Yaskawa INFORM job: SKRZYNIA_4040_90_STOPNI_10BR.JBI

/JOB
//NAME SKRZYNIA_4040_90_STOPNI_10BR
///FOLDERNAME 02-SKRZYNIE_JOBS
//POS
///NPOS 367,367,0,30,0,0
///TOOL 0
///POSTYPE PULSE
///PULSE
C00000=0,-52280,40443,0,6876,0
C00001=82314,-24956,17040,59626,-27382,6248
C00002=93910,-8625,17040,59626,-43355,6248
C00003=98846,-1061,-42166,80308,-57081,-16120
C00004=100452,6057,-48127,85711,-56704,-21322
C00005=96349,29000,-36127,85072,-63022,-26262
C00006=95580,33075,-33256,84644,-64024,-26851
C00007=94197,33846,-32020,85210,-63413,-26698
C00008=95580,33075,-33256,84644,-64024,-26851
C00009=94888,31114,-36362,85298,-63687,-27185
C00010=95580,33075,-33256,84644,-64024,-26851
C00011=95263,33142,-33256,84677,-63995,-26850
C00012=94634,33491,-32695,84935,-63717,-26781
C00013=94130,33776,-32235,85140,-63494,-26725
C00014=95104,32689,-33981,84829,-63917,-26928
C00015=94679,31503,-35865,85229,-63711,-27129
C00016=95263,33142,-33256,84677,-63995,-26850
C00017=95260,33144,-33256,84678,-63995,-26850
C00018=94650,33483,-32714,84929,-63727,-26783
C00019=94112,33789,-32223,85148,-63489,-26723
C00020=95084,32644,-34054,84845,-63909,-26937
C00021=94657,31449,-35950,85247,-63703,-27139
C00022=95260,33144,-33256,84678,-63995,-26850
C00023=95258,33145,-33257,84676,-63996,-26846
C00024=94953,33314,-32988,84801,-63862,-26812
C00025=94037,33833,-32158,85174,-63457,-26709
C00026=94978,32352,-34521,84941,-63860,-26983
C00027=94597,31295,-36193,85297,-63678,-27162
C00028=95258,33145,-33257,84676,-63996,-26846
C00029=95131,23090,-19879,77391,-65837,-18373
C00030=95120,22557,-18256,76776,-66108,-17621
C00031=94020,23265,-17262,77036,-65497,-17484
C00032=95120,22557,-18256,76776,-66108,-17621
C00033=94446,20406,-21237,77153,-65637,-17798
C00034=95120,22557,-18256,76776,-66108,-17621
C00035=95258,25631,32269,66559,-75499,-2416
C00036=95045,25799,32513,66531,-75379,-2372
C00037=94321,26382,33365,66429,-74973,-2219
C00038=95048,24784,31042,66584,-75290,-2483
C00039=94601,23046,28557,66633,-74859,-2609
C00040=95258,25631,32269,66559,-75499,-2416
C00041=98976,20539,9939,91612,-77544,-12443
C00042=98663,19916,6255,96113,-78269,-14194
C00043=97696,20512,7070,96235,-77611,-14191
C00044=98663,19916,6255,96113,-78269,-14194
C00045=98223,18195,3936,96233,-78026,-14357
C00046=98663,19916,6255,96113,-78269,-14194
C00047=97427,28150,42411,98154,-74759,-5932
C00048=97263,29860,47728,98172,-74140,-4881
C00049=96724,30318,48431,98088,-73756,-4848
C00050=97263,29860,47728,98172,-74140,-4881
C00051=96934,28259,45288,98260,-74017,-5126
C00052=97263,29860,47728,98172,-74140,-4881
C00053=94584,-1413,-17679,107543,-63249,-17346
C00054=98313,-6448,-37250,118963,-73755,-22159
C00055=78553,-42873,-65341,123231,-58560,-22541
C00056=78553,-42984,-66830,123659,-59131,-22943
C00057=97528,-2571,-34675,119478,-73963,-22751
C00058=99837,29570,44224,93766,-77824,-5891
C00059=98826,26629,36097,93853,-77239,-6316
C00060=97856,27338,37141,93774,-76562,-6265
C00061=98826,26629,36097,93853,-77239,-6316
C00062=98480,25016,33743,93919,-77053,-6522
C00063=98826,26629,36097,93853,-77239,-6316
C00064=98236,-3223,-2089,95569,-57848,-9600
C00065=99665,-7201,-6146,95388,-58784,-9416
C00066=48287,-55324,-44178,47560,-5470,10915
C00067=48287,-44591,-17414,16172,-14532,25809
C00068=85348,-13130,13838,41209,-47455,8220
C00069=99199,18818,35660,68259,-73735,-6208
C00070=95720,15423,18785,70454,-68603,-10022
C00071=95720,15423,18785,70454,-68603,-10022
C00072=97055,28839,36684,71776,-79389,-10554
C00073=95990,29701,37981,71658,-78759,-10350
C00074=97107,29731,38027,71793,-79947,-10506
C00075=96750,29830,38178,71892,-80905,-10618
C00076=97107,29731,38027,71793,-79947,-10506
C00077=97055,28839,36684,71776,-79389,-10554
C00078=97055,28839,36684,71776,-79389,-10554
C00079=96028,29668,37934,71662,-78782,-10355
C00080=97055,28839,36684,71776,-79389,-10554
C00081=96569,26658,33449,71833,-78910,-10776
C00082=97055,28839,36684,71776,-79389,-10554
C00083=97055,28839,36684,71776,-79389,-10554
C00084=97055,28839,36684,71776,-79389,-10554
C00085=96073,29634,37879,71669,-78808,-10363
C00086=97055,28839,36684,71776,-79389,-10554
C00087=96556,26588,33346,71835,-78895,-10784
C00088=97055,28839,36684,71776,-79389,-10554
C00089=98688,24309,19320,80205,-78471,-15843
C00090=97055,28839,36684,71776,-79389,-10554
C00091=96070,29634,37881,71667,-78806,-10365
C00092=97055,28839,36684,71776,-79389,-10554
C00093=96542,26531,33264,71837,-78884,-10788
C00094=97055,28839,36684,71776,-79389,-10554
C00095=99365,31341,48046,89916,-78663,6818
C00096=99073,32081,50196,92103,-78109,9106
C00097=98192,32828,51372,91957,-77498,9198
C00098=99073,32081,50196,92103,-78109,9106
C00099=98754,30342,47494,92168,-77945,8838
C00100=99073,32081,50196,92103,-78109,9106
C00101=99780,4859,-8097,97657,-68809,-987
C00102=97427,-15161,-48802,114933,-63377,-9928
C00103=58629,-63760,-77671,121137,-32820,-9668
C00104=58629,-61479,-68873,115361,-30519,-6465
C00105=99951,-8451,-34696,112012,-62700,-7410
C00106=99840,9300,10356,88107,-67494,6780
C00107=99532,23468,17388,90363,-79729,4530
C00108=98411,24191,18413,90419,-78957,4585
C00109=99532,23468,17388,90363,-79729,4530
C00110=99197,22008,15342,90436,-79518,4380
C00111=99532,23468,17388,90363,-79729,4530
C00112=99181,28193,42168,91916,-77030,2884
C00113=98696,27952,42277,91826,-76680,2991
C00114=97999,28483,43076,91734,-76199,3043
C00115=98696,27952,42277,91826,-76680,2991
C00116=98413,26578,40229,91881,-76520,2806
C00117=98696,27952,42277,91826,-76680,2991
C00118=97580,27630,40848,98508,-75244,1367
C00119=97580,27630,40848,98508,-75244,1367
C00120=96916,28152,41628,98436,-74775,1393
C00121=97580,27630,40848,98508,-75244,1367
C00122=97284,26265,38823,98576,-75120,1175
C00123=97580,27630,40848,98508,-75244,1367
C00124=99733,13297,3830,102164,-74334,-5956
C00125=98571,-14980,-17267,89913,-51486,-3548
C00126=44618,-53328,-38563,-7720,-11978,41868
C00127=44299,-51091,-32799,-7549,-14278,41753
///LIMIT ON
C00128=42729,-66511,10542,-1460,2814,7972
C00129=39797,-63802,12228,-1730,2225,8862
///LIMIT OFF
C00130=0,-43112,23163,-32261,-40956,-29092
C00131=50509,-19000,10610,51503,-15997,-61182
C00132=51153,-18191,11234,52953,-16222,-61812
C00133=49506,-16603,12499,51322,-15186,-61219
C00134=50699,-16390,12671,53298,-15774,-62041
C00135=50704,-18403,11069,52157,-16018,-61478
C00136=50704,-18403,11069,52157,-16018,-61478
C00137=51011,-18259,11181,52703,-16157,-61707
C00138=49372,-16676,12437,51065,-15128,-61110
C00139=50855,-16321,12727,53567,-15849,-62152
C00140=50704,-18403,11069,52157,-16018,-61478
C00141=50704,-18403,11069,52157,-16018,-61478
C00142=51194,-17966,11787,52443,-16367,-61556
C00143=49641,-16469,12982,50879,-15396,-60984
C00144=51159,-16110,13274,53409,-16135,-62034
C00145=51194,-19029,8982,55593,-15729,-63095
C00146=51005,-17995,11387,52847,-16122,-61778
C00147=51030,-17982,11395,52891,-16135,-61798
C00148=49666,-16664,12446,51542,-15278,-61306
C00149=51234,-16283,12753,54139,-16047,-62382
C00150=51030,-17982,11395,52891,-16135,-61798
C00151=51030,-17982,11395,52891,-16135,-61798
C00152=51056,-17951,11420,52949,-16145,-61823
C00153=49507,-16445,12622,51407,-15172,-61259
C00154=51212,-15994,12989,54262,-16005,-62444
C00155=51056,-17951,11420,52949,-16145,-61823
C00156=50945,-18019,11363,52741,-16103,-61737
C00157=51451,-18380,9957,55416,-15976,-62984
C00158=49638,-16617,11364,53777,-14815,-62399
C00159=51249,-16205,11700,56405,-15635,-63491
C00160=50945,-18019,11363,52741,-16103,-61737
C00161=50945,-18019,11363,52741,-16103,-61737
C00162=51751,-18888,8325,57986,-15754,-64205
C00163=49901,-17096,9744,56519,-14545,-63700
C00164=51443,-16713,10055,58931,-15359,-64698
C00165=50945,-18019,11363,52741,-16103,-61737
C00166=50945,-18019,11363,52741,-16103,-61737
C00167=51752,-17629,11670,54137,-16475,-62321
C00168=49778,-15710,13222,52239,-15234,-61634
C00169=51536,-15216,13634,55124,-16102,-62830
C00170=50945,-18019,11363,52741,-16103,-61737
C00171=50028,-22953,-3957,22347,-31919,-54220
C00172=50556,-22259,-3444,23037,-31901,-54554
C00173=48685,-20311,-1961,21193,-31011,-53711
C00174=50316,-19877,-1623,23110,-31344,-54618
C00175=49456,-22793,-3840,21729,-31736,-53932
C00176=49763,-25421,-36239,24565,-26935,-60445
C00177=49763,-25421,-36239,24565,-26935,-60445
C00178=47682,-22631,-34091,22709,-25786,-59390
C00179=49411,-21994,-33587,24802,-26153,-60557
C00180=49763,-25421,-36239,24565,-26935,-60445
C00181=50713,-12366,-58367,41124,-17813,-74400
C00182=50531,-11018,-57111,41258,-17631,-74434
C00183=49339,-9106,-55286,40470,-17030,-73839
C00184=50327,-8799,-54988,41498,-17395,-74518
C00185=50078,-11370,-57441,40744,-17481,-74102
C00186=49763,-25421,-36239,24565,-26935,-60445
C00187=49426,-25689,-5908,21254,-32432,-53672
C00188=45389,-28224,4312,35967,-15579,-54278
C00189=40154,-51179,-915,24203,-8234,-36524
C00190=0,-52280,40443,0,6876,0
C00191=21882,-20913,35982,82443,-51729,-53498
C00192=-23487,-14810,34938,67734,-39470,-58782
C00193=1657,-52280,40443,-304,6876,209
C00194=80083,-25473,16734,55938,-25627,7512
C00195=92674,-9533,16184,58080,-41894,6874
C00196=98391,-2369,-43566,80825,-55961,-16033
C00197=100022,4785,-49618,86526,-55706,-21348
C00198=95373,33537,-36121,86560,-63232,-28029
C00199=93881,36038,-32437,85059,-64562,-27761
C00200=93867,33044,-30650,83528,-64743,-25992
C00201=94930,31411,-33227,84334,-64171,-26252
C00202=94930,31411,-33227,84334,-64171,-26252
C00203=93474,31409,-33627,85103,-63552,-26381
C00204=93474,31409,-33627,85103,-63552,-26381
C00205=96539,31728,-33125,83558,-64961,-26367
C00206=95609,19235,-3385,72159,-68881,-11456
C00207=93675,20756,-1492,72153,-69304,-11461
C00208=93706,20835,-1296,72059,-69329,-11411
C00209=95041,22056,296,71883,-70234,-11460
C00210=95041,22056,296,71883,-70234,-11460
C00211=93716,20674,-1606,72153,-69328,-11471
C00212=93749,20787,-1450,72141,-69355,-11463
C00213=95041,22056,296,71883,-70234,-11460
C00214=95041,22056,296,71883,-70234,-11460
C00215=93853,20645,-1646,72134,-69414,-11487
C00216=93701,20690,-1585,72152,-69318,-11471
C00217=95606,21673,-233,71830,-70568,-11545
C00218=95936,-8790,-36169,76308,-52611,-10237
C00219=87381,-35372,-46042,66676,-50803,-1891
C00220=84950,-62287,8062,38288,-37295,1216
C00221=1657,-52280,40443,-304,6876,209
C00222=1657,-52280,40443,-304,6876,209
C00223=-4811,-36310,24637,-49210,-33845,-31988
C00224=41748,-30202,7105,17690,-22932,-42913
C00225=41748,-30202,7105,17690,-22932,-42913
C00226=49037,-21406,10886,33705,-21312,-49933
C00227=57938,-18196,5914,66765,-23183,-68504
C00228=62071,-18819,1330,80566,-26873,-76175
C00229=48249,-23742,8050,33819,-21114,-50004
C00230=-4811,-36310,24637,-49210,-33845,-31988
C00231=1657,-52280,40443,-304,6876,209
C00232=1613,-52280,40443,-296,6876,203
C00233=73560,-62084,7826,28695,-34737,3666
C00234=88377,-34186,-45291,67238,-52212,-2442
C00235=96528,-7533,-34932,76119,-53878,-10439
C00236=100432,21324,12575,83706,-77956,-7498
C00237=98573,22459,14150,83808,-76714,-7352
C00238=97947,26162,19403,83388,-79252,-7038
C00239=97765,26055,19247,83403,-79128,-7046
C00240=99338,18438,8643,84272,-74238,-7648
C00241=98912,19503,1370,96695,-78255,-12346
C00242=97381,18031,1012,96808,-77106,-12025
C00243=97381,18801,8446,95887,-76370,-9901
C00244=100328,20132,10252,95491,-78302,-9647
C00245=98154,32660,54986,101992,-72792,-1753
C00246=94873,38042,64057,104358,-72377,-1226
C00247=94755,38516,64855,104290,-72246,-1148
C00248=94753,45242,81749,102352,-70375,1916
C00249=96613,30369,38748,107128,-77305,-6302
C00250=98457,3518,-7444,102098,-66291,-11392
C00251=98781,-10331,-34310,114047,-66123,-16914
C00252=78936,-45022,-59687,116093,-50330,-16267
C00253=58820,-39124,10926,53325,-41870,3759
C00254=0,-52280,40443,0,6876,0
C00255=0,-36700,24612,-42871,-31823,-33862
C00256=44403,-30110,7154,24155,-23805,-45557
C00257=48366,-23967,9999,33441,-23050,-49710
C00258=57059,-21871,4355,62840,-24072,-66406
C00259=62664,-18498,1251,81512,-27948,-78180
C00260=58407,3196,49521,75767,-22763,-71356
C00261=56068,8902,60102,77374,-19708,-71368
C00262=52721,-13182,18231,110850,-19193,-88536
C00263=47073,-34549,9488,27883,-30316,-51458
C00264=0,-52247,40504,0,6859,0
C00265=41126,-41934,51032,-5894,-46731,13127
C00266=87376,-42070,-11985,58546,-50710,87
C00267=101177,-2604,23124,67435,-62482,198
C00268=97923,11434,18635,75872,-68057,-4429
C00269=99135,26942,27967,80896,-80067,-11
C00270=97959,27246,28410,80885,-79279,71
C00271=97910,25581,20036,81620,-78756,-2039
C00272=99054,25606,22085,82627,-78975,-1891
C00273=98877,27968,32487,76173,-79945,2468
C00274=95369,26181,23160,71095,-76769,901
C00275=95369,28262,32501,70203,-78207,3099
C00276=100802,24456,20984,80151,-80320,-697
C00277=99662,22785,17568,82066,-77607,-1267
C00278=97757,25456,21360,81884,-78797,-1037
C00279=97789,25433,21327,81884,-78819,-1041
C00280=99676,21999,16470,82145,-76972,-1318
C00281=97441,-6012,-18634,86114,-58345,-2339
C00282=92377,-33385,-41303,83059,-36844,1354
C00283=79425,-37128,-15462,51820,-35721,18807
C00284=43180,-50572,-20637,6552,-29302,38834
///LIMIT ON
C00285=37721,-67612,11381,1325,-438,7850
///LIMIT OFF
C00286=37164,-60659,6466,13301,-5027,-19773
C00287=45362,-39990,2831,27538,-17767,-40935
C00288=55315,-20486,12421,43917,-25084,-54085
C00289=61687,-17127,4357,78253,-26449,-75506
C00290=66887,-15221,5723,82563,-32969,-76938
C00291=53534,-30170,6270,37667,-26637,-51098
C00292=41180,-61187,4729,17280,-8498,-23442
C00293=0,-52280,40443,0,6876,0
C00294=0,-52280,40443,0,6876,0
///LIMIT ON
C00295=37721,-67612,11381,1325,-438,7850
///LIMIT OFF
C00296=43180,-50572,-20637,6552,-29302,38834
C00297=79425,-37128,-15462,51820,-35721,18807
C00298=92377,-33385,-41303,83059,-36844,1354
C00299=100252,-4949,-17551,85890,-60241,-2391
C00300=99662,22785,17568,82066,-77607,-1267
C00301=98003,26711,23176,81782,-79695,-932
C00302=98187,26766,23256,81772,-79821,-932
C00303=99662,22785,17568,82066,-77607,-1267
C00304=99662,22785,17568,82066,-77607,-1267
C00305=97671,26258,22515,81825,-79282,-965
C00306=97727,26283,22551,81822,-79321,-966
C00307=99662,22785,17568,82066,-77607,-1267
C00308=99171,25371,27709,97207,-78195,-1592
C00309=97098,23330,25144,97300,-76842,-1817
C00310=97098,25842,34993,96283,-76010,469
C00311=99772,20639,8352,98678,-80464,-6065
C00312=98552,-10425,-57317,115530,-68576,-16387
C00313=72212,-55568,-87372,121854,-47773,-15081
C00314=43180,-50572,-20637,6552,-29302,38834
///LIMIT ON
C00315=37721,-67612,11381,1325,-438,7850
///LIMIT OFF
C00316=0,-52280,40443,0,6876,0
C00317=0,-52280,40443,0,6876,0
///LIMIT ON
C00318=23708,-46776,23536,16027,-4787,-19738
///LIMIT OFF
C00319=50917,-40459,4132,34421,-18173,-42391
C00320=55315,-20486,12421,43917,-25084,-54085
C00321=52021,-27344,-11614,25442,-32756,-51822
C00322=62388,-19076,-7315,47741,-37100,-57915
C00323=60492,-23043,-43968,60514,-28343,-68592
C00324=52021,-27344,-11614,25442,-32756,-51822
C00325=50917,-40459,4132,34421,-18173,-42391
C00326=56351,-28617,-8977,50177,-24220,-59041
C00327=61013,-25727,-20437,91852,-25479,-87385
C00328=68741,-23000,-19911,95900,-36007,-87783
C00329=59870,-32730,-20784,77712,-26701,-76039
C00330=36994,-41399,-15582,14937,-21377,-43241
C00331=31287,-69981,-10850,7253,-6843,-20996
C00332=19644,-57271,30737,863,5243,-2499
C00333=0,-52280,40443,0,6876,0
C00334=0,-52280,40443,0,6876,0
///LIMIT ON
C00335=37721,-67612,11381,1325,-438,7850
///LIMIT OFF
C00336=43180,-50572,-20637,6552,-29302,38834
C00337=92325,-17806,9716,57334,-44195,17168
C00338=83562,-2075,23934,52242,-47081,17120
C00339=81926,-4528,18929,54087,-44625,16400
C00340=98156,27605,40467,74304,-79249,6093
C00341=97389,28448,36068,78537,-79231,3814
C00342=97907,24801,21502,85617,-78711,-660
C00343=99547,21785,17244,85874,-76675,-945
C00344=99107,21615,15088,95660,-77501,-3171
C00345=97330,21661,23948,94493,-75452,-401
C00346=97330,25174,37197,92971,-74702,2673
C00347=100285,22853,27662,91564,-77234,921
C00348=95045,29770,44207,110893,-72615,-445
C00349=92602,30098,46290,110515,-70628,-245
C00350=91321,34137,56434,112423,-68257,619
C00351=92127,32273,50247,113174,-70001,-486
C00352=99547,27249,39584,83596,-77197,4391
C00353=85644,-16652,-26140,89995,-40279,-1638
C00354=96357,-21723,-30363,88205,-47532,-883
C00355=98913,1421,32623,59426,-59934,14740
C00356=68865,-35989,-5252,49829,-38105,21179
C00357=80632,-38079,-20908,64053,-45216,12949
C00358=43180,-50572,-20637,6552,-29302,38834
C00359=50917,-40459,4132,34421,-18173,-42391
C00360=55315,-20486,12421,43917,-25084,-54085
C00361=52609,-18323,14042,41333,-23544,-53138
C00362=70054,-15959,-1295,94448,-37577,-86566
C00363=61757,-17157,6384,73937,-27308,-72117
C00364=37618,-28118,7425,14704,-21495,-41826
C00365=31287,-69981,-10850,7253,-6843,-20996
C00366=0,-52280,40443,0,6876,0
BC00000=376110
BC00001=352964
BC00002=352964
BC00003=352964
BC00004=352964
BC00005=352964
BC00006=352964
BC00007=352964
BC00008=352964
BC00009=352964
BC00010=352964
BC00011=399066
BC00012=399066
BC00013=399066
BC00014=399066
BC00015=399066
BC00016=399066
BC00017=445276
BC00018=445276
BC00019=445276
BC00020=445276
BC00021=445276
BC00022=445276
BC00023=491380
BC00024=491380
BC00025=491380
BC00026=491380
BC00027=491380
BC00028=491380
BC00029=477558
BC00030=476336
BC00031=476336
BC00032=476336
BC00033=476336
BC00034=476336
BC00035=467227
BC00036=467227
BC00037=467227
BC00038=467227
BC00039=467227
BC00040=467227
BC00041=479694
BC00042=482001
BC00043=482001
BC00044=482001
BC00045=482001
BC00046=482001
BC00047=469388
BC00048=468082
BC00049=468082
BC00050=468082
BC00051=468082
BC00052=468082
BC00053=467166
BC00054=467166
BC00055=467166
BC00056=581600
BC00057=581600
BC00058=528199
BC00059=528202
BC00060=528202
BC00061=528202
BC00062=528202
BC00063=528202
BC00064=531560
BC00065=531560
BC00066=512089
BC00067=606955
BC00068=621951
BC00069=621951
BC00070=621951
BC00071=621951
BC00072=621951
BC00073=621951
BC00074=621951
BC00075=621951
BC00076=621951
BC00077=645037
BC00078=645037
BC00079=645037
BC00080=645037
BC00081=645037
BC00082=645037
BC00083=691109
BC00084=691109
BC00085=691109
BC00086=691109
BC00087=691109
BC00088=691109
BC00089=714197
BC00090=714197
BC00091=714197
BC00092=714197
BC00093=714197
BC00094=714197
BC00095=704400
BC00096=703157
BC00097=703157
BC00098=703157
BC00099=703157
BC00100=703157
BC00101=703157
BC00102=713115
BC00103=713115
BC00104=805551
BC00105=805551
BC00106=781418
BC00107=793824
BC00108=793824
BC00109=793824
BC00110=793824
BC00111=793824
BC00112=808984
BC00113=808984
BC00114=808984
BC00115=808984
BC00116=808984
BC00117=808984
BC00118=829368
BC00119=829368
BC00120=829368
BC00121=829368
BC00122=829368
BC00123=829368
BC00124=829627
BC00125=821657
BC00126=814103
BC00127=795686
BC00128=693498
BC00129=688280
BC00130=719629
BC00131=797458
BC00132=797458
BC00133=797458
BC00134=797458
BC00135=797458
BC00136=736016
BC00137=736016
BC00138=736016
BC00139=736016
BC00140=736016
BC00141=674586
BC00142=674586
BC00143=674586
BC00144=674586
BC00145=674586
BC00146=613184
BC00147=613184
BC00148=613184
BC00149=613184
BC00150=613184
BC00151=555022
BC00152=555022
BC00153=555022
BC00154=555022
BC00155=555022
BC00156=490298
BC00157=490298
BC00158=490298
BC00159=490298
BC00160=490298
BC00161=428826
BC00162=428826
BC00163=428826
BC00164=428826
BC00165=428826
BC00166=367374
BC00167=367374
BC00168=367374
BC00169=367374
BC00170=367374
BC00171=367378
BC00172=367378
BC00173=367378
BC00174=367378
BC00175=367378
BC00176=367378
BC00177=367378
BC00178=367378
BC00179=367378
BC00180=367378
BC00181=367378
BC00182=367378
BC00183=367378
BC00184=367378
BC00185=367378
BC00186=367378
BC00187=367378
BC00188=367374
BC00189=441050
BC00190=441050
BC00191=743708
BC00192=782128
BC00193=352964
BC00194=352964
BC00195=352964
BC00196=406723
BC00197=352964
BC00198=352964
BC00199=352964
BC00200=353556
BC00201=353556
BC00202=391964
BC00203=400107
BC00204=389591
BC00205=400107
BC00206=381081
BC00207=388817
BC00208=381081
BC00209=388818
BC00210=427169
BC00211=434877
BC00212=427169
BC00213=427169
BC00214=450237
BC00215=457913
BC00216=450237
BC00217=450041
BC00218=450041
BC00219=450041
BC00220=450041
BC00221=450041
BC00222=400994
BC00223=490644
BC00224=563016
BC00225=563016
BC00226=563016
BC00227=563016
BC00228=624476
BC00229=624476
BC00230=490644
BC00231=400994
BC00232=402304
BC00233=450041
BC00234=450041
BC00235=498778
BC00236=451598
BC00237=451598
BC00238=459362
BC00239=451598
BC00240=459288
BC00241=484574
BC00242=484574
BC00243=484574
BC00244=484574
BC00245=464718
BC00246=464718
BC00247=464718
BC00248=469790
BC00249=469790
BC00250=467718
BC00251=475246
BC00252=427384
BC00253=476890
BC00254=492251
BC00255=720637
BC00256=795617
BC00257=801528
BC00258=805368
BC00259=808796
BC00260=777283
BC00261=777283
BC00262=777285
BC00263=760893
BC00264=538671
BC00265=564292
BC00266=544905
BC00267=523419
BC00268=548184
BC00269=573245
BC00270=573245
BC00271=573245
BC00272=569148
BC00273=617841
BC00274=629475
BC00275=629475
BC00276=631879
BC00277=634993
BC00278=633229
BC00279=640937
BC00280=640937
BC00281=640937
BC00282=640937
BC00283=640937
BC00284=640937
BC00285=640937
BC00286=469376
BC00287=406602
BC00288=315730
BC00289=315725
BC00290=377231
BC00291=377231
BC00292=431999
BC00293=431999
BC00294=640937
BC00295=640937
BC00296=640937
BC00297=640937
BC00298=640937
BC00299=640937
BC00300=679258
BC00301=679258
BC00302=687013
BC00303=679258
BC00304=702338
BC00305=702338
BC00306=710018
BC00307=702338
BC00308=711372
BC00309=711372
BC00310=711372
BC00311=711372
BC00312=723912
BC00313=723912
BC00314=703131
BC00315=640937
BC00316=640937
BC00317=492251
BC00318=483911
BC00319=372992
BC00320=315730
BC00321=315730
BC00322=315730
BC00323=315730
BC00324=315730
BC00325=421515
BC00326=465804
BC00327=465238
BC00328=526388
BC00329=526326
BC00330=526236
BC00331=526236
BC00332=526236
BC00333=526236
BC00334=640937
BC00335=640937
BC00336=792907
BC00337=785422
BC00338=785422
BC00339=785422
BC00340=808786
BC00341=808610
BC00342=816482
BC00343=816482
BC00344=831767
BC00345=831767
BC00346=831767
BC00347=831767
BC00348=812640
BC00349=812640
BC00350=812640
BC00351=812640
BC00352=814454
BC00353=818927
BC00354=798802
BC00355=772424
BC00356=743273
BC00357=702349
BC00358=657048
BC00359=664515
BC00360=684473
BC00361=684473
BC00362=684473
BC00363=745829
BC00364=745829
BC00365=650116
BC00366=650116
///POSTYPE BASE
///RECTAN
///RCONF 0,0,0,0,0,0,0,0,0,0,0,0,0,0,0,0,0,0,0,0,0,0,0,0
P00006=-2.449,0.031,8.825,0.0000,0.0000,0.0000
P00058=0.000,0.000,3.000,0.0000,0.0000,0.0000
///RCONF 1,0,0,0,0,0,0,0,0,0,0,0,0,0,0,0,0,0,0,0,0,0,0,0
P00300=-0.036,-1.505,2.318,0.0000,0.0000,0.0000
///RCONF 0,0,0,0,0,0,0,0,0,0,0,0,0,0,0,0,0,0,0,0,0,0,0,0
P00301=0.005,-4.708,-4.628,0.0000,0.0000,0.0000
P00302=0.052,-2.937,-4.426,0.0000,0.0000,0.0000
P00303=-0.004,-1.437,-4.584,0.0000,0.0000,0.0000
P00304=0.028,-1.666,-4.234,0.0000,0.0000,0.0000
P00305=-0.003,-1.920,-3.501,0.0000,0.0000,0.0000
P00306=0.015,-2.252,-3.054,0.0000,0.0000,0.0000
P00307=0.019,-2.151,-5.077,0.0000,0.0000,0.0000
P00308=-0.003,-2.092,-4.888,0.0000,0.0000,0.0000
P00309=-0.040,-2.205,-4.992,0.0000,0.0000,0.0000
P00310=-0.006,-2.490,-5.925,0.0000,0.0000,0.0000
P00311=-0.007,-2.079,-5.307,0.0000,0.0000,0.0000
P00312=-0.032,2.202,-7.632,0.0000,0.0000,0.0000
///RCONF 1,0,0,0,0,0,0,0,0,0,0,0,0,0,0,0,0,0,0,0,0,0,0,0
P00313=-0.088,1.055,2.110,0.0000,0.0000,0.0000
P00314=-0.055,1.752,1.634,0.0000,0.0000,0.0000
P00316=0.009,2.112,2.075,0.0000,0.0000,0.0000
P00317=-0.015,2.781,3.126,0.0000,0.0000,0.0000
///RCONF 0,0,0,0,0,0,0,0,0,0,0,0,0,0,0,0,0,0,0,0,0,0,0,0
P00351=13.563,-0.027,-0.653,0.0000,0.0000,0.0000
P00352=13.252,-0.027,-0.827,0.0000,0.0000,0.0000
P00353=10.971,-0.082,0.776,0.0000,0.0000,0.0000
P00354=-0.024,2.508,-1.824,0.0000,0.0000,0.0000
P00355=-0.001,2.528,-1.131,0.0000,0.0000,0.0000
P00356=-0.034,2.921,-0.262,0.0000,0.0000,0.0000
P00357=0.003,3.386,-0.091,0.0000,0.0000,0.0000
P00358=0.014,3.037,-0.020,0.0000,0.0000,0.0000
P00359=-0.005,2.731,0.912,0.0000,0.0000,0.0000
P00360=-0.011,3.412,0.438,0.0000,0.0000,0.0000
P00361=0.018,3.050,1.253,0.0000,0.0000,0.0000
//INST
///DATE 2025/03/25 09:39
///ATTR SC,RW
///GROUP1 RB1,BS1
NOP
CALL JOB:MOVE_INTO_TUNNEL
MOVJ C00000 BC00000 VJ=50.00
MOVJ C00001 BC00001 VJ=30.00
MOVJ C00002 BC00002 VJ=30.00
COMM MOVL C00003 BC00003 V=333.3
COMM MOVJ C00004 BC00004 VJ=30.00
COMM MOVL C00005 BC00005 V=500.0
COMM '------------------------
COMM 'W31.2
COMM '------------------------
COMM MOVL C00006 BC00006 V=166.7 PL=0
COMM REFP 3 C00007 BC00007
COMM CALL JOB:SEARCH-R1
COMM SET P0300 P0006
COMM SFTON P0300
COMM MOVL C00008 BC00008 V=66.7 PL=0
COMM REFP 3 C00009 BC00009
COMM CALL JOB:SEARCH-R1
COMM SET P0300 P0006
COMM SFTON P0300
COMM MOVL C00010 BC00010 V=166.7 PL=0
COMM SFTOF
COMM '------------------------
COMM 'W31.4
COMM '------------------------
COMM MOVL C00011 BC00011 V=666.7
COMM MOVL C00012 BC00012 V=83.3 PL=0
COMM REFP 3 C00013 BC00013
COMM CALL JOB:SEARCH-R1
COMM SET P0301 P0006
COMM SFTON P0301
COMM MOVL C00014 BC00014 V=166.7 PL=0
COMM REFP 3 C00015 BC00015
COMM CALL JOB:SEARCH-R1
COMM SET P0301 P0006
COMM SFTON P0301
COMM MOVL C00016 BC00016 V=166.7 PL=0
COMM SFTOF
'------------------------
'W31.6
'------------------------
MOVL C00017 BC00017 V=666.7
MOVL C00018 BC00018 V=83.3 PL=0
REFP 3 C00019 BC00019
CALL JOB:SEARCH-R1
SET P0302 P0006
SFTON P0302
MOVL C00020 BC00020 V=166.7 PL=0
REFP 3 C00021 BC00021
CALL JOB:SEARCH-R1
SET P0302 P0006
SFTON P0302
MOVL C00022 BC00022 V=250.0 PL=0
SFTOF
'------------------------
'W31.8
'------------------------
MOVL C00023 BC00023 V=666.7
MOVL C00024 BC00024 V=83.3 PL=0
REFP 3 C00025 BC00025
CALL JOB:SEARCH-R1
SET P0303 P0006
SFTON P0303
MOVL C00026 BC00026 V=166.7 PL=0
REFP 3 C00027 BC00027
CALL JOB:SEARCH-R1
SET P0303 P0006
SFTON P0303
MOVL C00028 BC00028 V=250.0 PL=0
SFTOF
'------------------------
'W31.9
'------------------------
MOVL C00029 BC00029 V=666.7
MOVL C00030 BC00030 V=83.3 PL=0
REFP 3 C00031 BC00031
CALL JOB:SEARCH-R1
SET P0304 P0006
SFTON P0304
MOVL C00032 BC00032 V=166.7 PL=0
REFP 3 C00033 BC00033
CALL JOB:SEARCH-R1
SET P0304 P0006
SFTON P0304
MOVL C00034 BC00034 V=250.0 PL=0
SFTOF
'------------------------
'W31.11
'------------------------
MOVL C00035 BC00035 V=666.7
MOVL C00036 BC00036 V=83.3 PL=0
REFP 3 C00037 BC00037
CALL JOB:SEARCH-R1
SET P0305 P0006
SFTON P0305
MOVL C00038 BC00038 V=166.7 PL=0
REFP 3 C00039 BC00039
CALL JOB:SEARCH-R1
SET P0305 P0006
SFTON P0305
MOVL C00040 BC00040 V=250.0 PL=0
SFTOF
'------------------------
'W31.13
'------------------------
MOVL C00041 BC00041 V=666.7
MOVL C00042 BC00042 V=166.7 PL=0
REFP 3 C00043 BC00043
CALL JOB:SEARCH-R1
SET P0306 P0006
SFTON P0306
MOVL C00044 BC00044 V=166.7 PL=0
REFP 3 C00045 BC00045
CALL JOB:SEARCH-R1
SET P0306 P0006
SFTON P0306
MOVL C00046 BC00046 V=250.0 PL=0
SFTOF
'------------------------
'W31.14
'------------------------
MOVL C00047 BC00047 V=666.7
MOVL C00048 BC00048 V=100.0 PL=0
REFP 3 C00049 BC00049
CALL JOB:SEARCH-R1
SET P0307 P0006
SFTON P0307
MOVL C00050 BC00050 V=166.7 PL=0
REFP 3 C00051 BC00051
CALL JOB:SEARCH-R1
SET P0307 P0006
SFTON P0307
MOVL C00052 BC00052 V=250.0 PL=0
SFTOF
'------------------------
MOVL C00053 BC00053 V=333.3
MOVL C00054 BC00054 V=333.3
MOVL C00055 BC00055 V=333.3
MOVL C00056 BC00056 V=666.7
MOVL C00057 BC00057 V=666.7
'W31.16
'------------------------
MOVL C00058 BC00058 V=666.7
MOVL C00059 BC00059 V=100.0 PL=0
REFP 3 C00060 BC00060
CALL JOB:SEARCH-R1
SET P0308 P0006
SFTON P0308
MOVL C00061 BC00061 V=166.7 PL=0
REFP 3 C00062 BC00062
CALL JOB:SEARCH-R1
SET P0308 P0006
SFTON P0308
MOVL C00063 BC00063 V=250.0 PL=0
SFTOF
MOVL C00064 BC00064 V=666.7
MOVL C00065 BC00065 V=666.7
MOVL C00066 BC00066 V=500.0 PL=1
MOVJ C00067 BC00067 VJ=60.00
MOVL C00068 BC00068 V=833.3 PL=0
MOVL C00069 BC00069 V=500.0 PL=0
MOVL C00070 BC00070 V=500.0 PL=0
'------------------------
'W31.18
'------------------------
MOVL C00071 BC00071 V=333.3 PL=0
SFTOF
MOVL C00072 BC00072 V=133.3 PL=0
REFP 3 C00073 BC00073
CALL JOB:SEARCH-R1
SET P0309 P0006
SFTON P0309
MOVL C00074 BC00074 V=166.7 PL=0
REFP 3 C00075 BC00075
CALL JOB:SEARCH-R1
SET P0309 P0006
SFTON P0309
MOVL C00076 BC00076 V=250.0 PL=0
SFTOF
'------------------------
'W31.19
'------------------------
MOVL C00077 BC00077 V=666.7
MOVL C00078 BC00078 V=100.0 PL=0
REFP 3 C00079 BC00079
CALL JOB:SEARCH-R1
SET P0310 P0006
SFTON P0310
MOVL C00080 BC00080 V=166.7 PL=0
REFP 3 C00081 BC00081
CALL JOB:SEARCH-R1
SET P0310 P0006
SFTON P0310
MOVL C00082 BC00082 V=250.0 PL=0
SFTOF
'------------------------
'W31.21
'------------------------
MOVL C00083 BC00083 V=666.7
MOVL C00084 BC00084 V=100.0 PL=0
REFP 3 C00085 BC00085
CALL JOB:SEARCH-R1
SET P0311 P0006
SFTON P0311
MOVL C00086 BC00086 V=166.7 PL=0
REFP 3 C00087 BC00087
CALL JOB:SEARCH-R1
SET P0311 P0006
SFTON P0311
MOVL C00088 BC00088 V=250.0 PL=0
SFTOF
'------------------------
'W31.22
'------------------------
MOVL C00089 BC00089 V=666.7
MOVL C00090 BC00090 V=100.0 PL=0
REFP 3 C00091 BC00091
CALL JOB:SEARCH-R1
SET P0312 P0006
SFTON P0312
MOVL C00092 BC00092 V=166.7 PL=0
REFP 3 C00093 BC00093
CALL JOB:SEARCH-R1
SET P0312 P0006
SFTON P0312
MOVL C00094 BC00094 V=250.0 PL=0
SFTOF
'------------------------
'W31.24
'------------------------
MOVL C00095 BC00095 V=666.7
MOVL C00096 BC00096 V=100.0 PL=0
REFP 3 C00097 BC00097
CALL JOB:SEARCH-R1
SET P0313 P0006
SFTON P0313
MOVL C00098 BC00098 V=166.7 PL=0
REFP 3 C00099 BC00099
CALL JOB:SEARCH-R1
SET P0313 P0006
SFTON P0313
MOVL C00100 BC00100 V=166.7 PL=0
SFTOF
MOVL C00101 BC00101 V=666.7
MOVL C00102 BC00102 V=666.7
MOVL C00103 BC00103 V=666.7
MOVL C00104 BC00104 V=666.7
MOVL C00105 BC00105 V=666.7
'------------------------
'W31.26
'------------------------
MOVL C00106 BC00106 V=666.7
MOVL C00107 BC00107 V=100.0 PL=0
REFP 3 C00108 BC00108
CALL JOB:SEARCH-R1
SET P0314 P0006
SFTON P0314
MOVL C00109 BC00109 V=166.7 PL=0
REFP 3 C00110 BC00110
CALL JOB:SEARCH-R1
SET P0314 P0006
SFTON P0314
MOVL C00111 BC00111 V=250.0 PL=0
SFTOF
'------------------------
'W31.29
'------------------------
MOVL C00112 BC00112 V=166.7
MOVL C00113 BC00113 V=100.0 PL=0
REFP 3 C00114 BC00114
CALL JOB:SEARCH-R1
SET P0316 P0006
SFTON P0316
MOVL C00115 BC00115 V=166.7 PL=0
REFP 3 C00116 BC00116
CALL JOB:SEARCH-R1
SET P0316 P0006
SFTON P0316
MOVL C00117 BC00117 V=250.0 PL=0
SFTOF
'------------------------
'W31.31
'------------------------
MOVL C00118 BC00118 V=250.0
MOVL C00119 BC00119 V=100.0 PL=0
REFP 3 C00120 BC00120
CALL JOB:SEARCH-R1
SET P0317 P0006
SFTON P0317
MOVL C00121 BC00121 V=166.7 PL=0
REFP 3 C00122 BC00122
CALL JOB:SEARCH-R1
SET P0317 P0006
SFTON P0317
MOVL C00123 BC00123 V=250.0 PL=0
SFTOF
'------------------------
'W31.32
'------------------------
MOVL C00124 BC00124 V=500.0
MOVL C00125 BC00125 V=500.0
MOVL C00126 BC00126 V=500.0
MOVL C00127 BC00127 V=666.7
MOVJ C00128 BC00128 VJ=80.00
MOVJ C00129 BC00129 VJ=80.00
MOVJ C00130 BC00130 VJ=50.00
'------------------------
'W214A L
'------------------------
MOVJ C00131 BC00131 VJ=30.00
MOVL C00132 BC00132 V=100.0 PL=0
REFP 3 C00133 BC00133
CALL JOB:SEARCH-R1
IMOV P0058 V=11.7
SET P0351 P0006
SFTON P0351
REFP 3 C00134 BC00134
CALL JOB:SEARCH-R1
SET P0351 P0006
SFTON P0351
MOVL C00135 BC00135 V=250.0 PL=0
SFTOF
'------------------------
'W219A P
'------------------------
MOVJ C00136 BC00136 VJ=40.00
MOVL C00137 BC00137 V=100.0 PL=0
REFP 3 C00138 BC00138
CALL JOB:SEARCH-R1
IMOV P0058 V=11.7
SET P0352 P0006
SFTON P0352
REFP 3 C00139 BC00139
CALL JOB:SEARCH-R1
SET P0352 P0006
SFTON P0352
MOVL C00140 BC00140 V=250.0 PL=0
SFTOF
'------------------------
'W219A L
'------------------------
MOVJ C00141 BC00141 VJ=50.00
MOVL C00142 BC00142 V=166.7 PL=0
REFP 3 C00143 BC00143
CALL JOB:SEARCH-R1
IMOV P0058 V=11.7
SET P0353 P0006
SFTON P0353
REFP 3 C00144 BC00144
CALL JOB:SEARCH-R1
SET P0353 P0006
SFTON P0353
MOVL C00145 BC00145 V=250.0 PL=0
SFTOF
'------------------------
'W213A P
'------------------------
MOVJ C00146 BC00146 VJ=60.00
MOVL C00147 BC00147 V=166.7 PL=0
REFP 3 C00148 BC00148
CALL JOB:SEARCH-R1
IMOV P0058 V=11.7
SET P0354 P0006
SFTON P0354
REFP 3 C00149 BC00149
CALL JOB:SEARCH-R1
SET P0354 P0006
SFTON P0354
MOVL C00150 BC00150 V=250.0 PL=0
SFTOF
'------------------------
'W213A L
'------------------------
MOVJ C00151 BC00151 VJ=50.00
MOVL C00152 BC00152 V=166.7 PL=0
REFP 3 C00153 BC00153
CALL JOB:SEARCH-R1
IMOV P0058 V=11.7
SET P0355 P0006
SFTON P0355
REFP 3 C00154 BC00154
CALL JOB:SEARCH-R1
SET P0355 P0006
SFTON P0355
MOVL C00155 BC00155 V=250.0 PL=0
SFTOF
'------------------------
'W218A P
'------------------------
MOVJ C00156 BC00156 VJ=60.00
MOVL C00157 BC00157 V=166.7 PL=0
REFP 3 C00158 BC00158
CALL JOB:SEARCH-R1
IMOV P0058 V=11.7
SET P0356 P0006
SFTON P0356
REFP 3 C00159 BC00159
CALL JOB:SEARCH-R1
SET P0356 P0006
SFTON P0356
MOVL C00160 BC00160 V=250.0 PL=0
SFTOF
'------------------------
'W218A L
'------------------------
MOVJ C00161 BC00161 VJ=60.00
MOVL C00162 BC00162 V=166.7 PL=0
REFP 3 C00163 BC00163
CALL JOB:SEARCH-R1
IMOV P0058 V=11.7
SET P0357 P0006
SFTON P0357
REFP 3 C00164 BC00164
CALL JOB:SEARCH-R1
SET P0357 P0006
SFTON P0357
MOVL C00165 BC00165 V=250.0 PL=0
SFTOF
'------------------------
'W215A P
'------------------------
MOVJ C00166 BC00166 VJ=60.00
MOVL C00167 BC00167 V=166.7 PL=0
REFP 3 C00168 BC00168
CALL JOB:SEARCH-R1
IMOV P0058 V=11.7
SET P0358 P0006
SFTON P0358
REFP 3 C00169 BC00169
CALL JOB:SEARCH-R1
SET P0358 P0006
SFTON P0358
MOVL C00170 BC00170 V=250.0 PL=0
SFTOF
'------------------------
'W215A L
'------------------------
MOVL C00171 BC00171 V=666.7
MOVL C00172 BC00172 V=166.7 PL=0
REFP 3 C00173 BC00173
CALL JOB:SEARCH-R1
IMOV P0058 V=11.7
SET P0359 P0006
SFTON P0359
REFP 3 C00174 BC00174
CALL JOB:SEARCH-R1
SET P0359 P0006
SFTON P0359
MOVL C00175 BC00175 V=66.7 PL=0
SFTOF
COMM '------------------------
COMM 'W217A P
COMM '------------------------
COMM MOVL C00176 BC00176 V=666.7
COMM MOVL C00177 BC00177 V=166.7 PL=0
COMM REFP 3 C00178 BC00178
COMM CALL JOB:SEARCH-R1
COMM IMOV P0058 V=11.7
COMM SET P0360 P0006
COMM SFTON P0360
COMM REFP 3 C00179 BC00179
COMM CALL JOB:SEARCH-R1
COMM SET P0360 P0006
COMM SFTON P0360
COMM MOVL C00180 BC00180 V=250.0 PL=0
COMM SFTOF
COMM '------------------------
COMM 'W217A L
COMM '------------------------
COMM MOVL C00181 BC00181 V=666.7
COMM MOVL C00182 BC00182 V=166.7 PL=0
COMM REFP 3 C00183 BC00183
COMM CALL JOB:SEARCH-R1
COMM IMOV P0058 V=11.7
COMM SET P0361 P0006
COMM SFTON P0361
COMM REFP 3 C00184 BC00184
COMM CALL JOB:SEARCH-R1
COMM SET P0361 P0006
COMM SFTON P0361
COMM MOVL C00185 BC00185 V=250.0 PL=0
COMM SFTOF
COMM MOVL C00186 BC00186 V=666.7
COMM MOVL C00187 BC00187 V=833.3
MOVL C00188 BC00188 V=833.3
MOVJ C00189 BC00189 VJ=70.00
MOVJ C00190 BC00190 VJ=80.00
MOVJ C00191 BC00191 VJ=50.00
MOVJ C00192 BC00192 VJ=80.00
CALL JOB:FRONT_SEARCH_90ST-1_4040
MOVJ C00193 BC00193 VJ=50.00
MOVJ C00194 BC00194 VJ=40.00
MOVJ C00195 BC00195 VJ=40.00
MOVL C00196 BC00196 V=500.0
COMM MOVJ C00197 BC00197 VJ=30.00
COMM '------------------------
COMM 'W31.2
COMM '------------------------
COMM SFTON P0300
COMM MOVL C00198 BC00198 V=500.0
COMM MOVL C00199 BC00199 V=133.3 PL=0
COMM MACRO1 MJ#(0) ARGF10
COMM ARCON
COMM MOVL C00200 BC00200 V=10.8
COMM ARCOF
COMM MOVL C00201 BC00201 V=250.0
COMM SFTOF
COMM '------------------------
COMM 'W31.4
COMM '------------------------
COMM SFTON P0301
COMM MOVL C00202 BC00202 V=500.0
COMM MOVL C00203 BC00203 V=166.7
COMM MACRO1 MJ#(0) ARGF10
COMM ARCON
COMM MOVL C00204 BC00204 V=10.8
COMM ARCOF
COMM MOVL C00205 BC00205 V=250.0
COMM SFTOF
'------------------------
'W31.6
'------------------------
SFTON P0302
MOVL C00206 BC00206 V=500.0
MOVL C00207 BC00207 V=166.7 PL=0
MACRO1 MJ#(0) ARGF10
ARCON
MOVL C00208 BC00208 V=10.8
ARCOF
MOVL C00209 BC00209 V=166.7
SFTOF
'------------------------
'W31.8
'------------------------
SFTON P0303
MOVL C00210 BC00210 V=500.0
MOVL C00211 BC00211 V=166.7 PL=0
MACRO1 MJ#(0) ARGF10
ARCON
MOVL C00212 BC00212 V=10.8
ARCOF
MOVL C00213 BC00213 V=166.7
SFTOF
'------------------------
'W31.9
'------------------------
SFTON P0304
MOVL C00214 BC00214 V=500.0
MOVL C00215 BC00215 V=166.7 PL=0
MACRO1 MJ#(0) ARGF10
ARCON
MOVL C00216 BC00216 V=10.8
ARCOF
MOVL C00217 BC00217 V=166.7
SFTOF
MOVL C00218 BC00218 V=500.0
MOVL C00219 BC00219 V=666.7
MOVJ C00220 BC00220 VJ=30.00
MOVJ C00221 BC00221 VJ=50.00
MOVJ C00222 BC00222 VJ=50.00
MOVJ C00223 BC00223 VJ=50.00
MOVJ C00224 BC00224 VJ=50.00
MOVL C00225 BC00225 V=166.7
'------------------------
'W213A
'------------------------
SFTON P0355
MOVL C00226 BC00226 V=500.0
MOVL C00227 BC00227 V=166.7 PL=0
MACRO1 MJ#(0) ARGF9
ARCON
SFTOF
SFTON P0354
MOVL C00228 BC00228 V=11.7
ARCOF
MOVL C00229 BC00229 V=166.7
SFTOF
MOVJ C00230 BC00230 VJ=50.00
MOVJ C00231 BC00231 VJ=80.00
MOVJ C00232 BC00232 VJ=10.00
MOVJ C00233 BC00233 VJ=40.00
MOVJ C00234 BC00234 VJ=40.00
MOVJ C00235 BC00235 VJ=30.00
MOVJ C00236 BC00236 VJ=30.00
'5.5.1
'------------------------
'W31.11
'------------------------
SFTON P0305
MOVL C00237 BC00237 V=333.3
MOVL C00238 BC00238 V=166.7
MACRO1 MJ#(0) ARGF10
ARCON
MOVL C00239 BC00239 V=10.8
ARCOF
MOVL C00240 BC00240 V=166.7
SFTOF
'------------------------
'W31.13
'------------------------
SFTON P0306
MOVL C00241 BC00241 V=333.3
MOVL C00242 BC00242 V=166.7
ARCON
MOVL C00243 BC00243 V=10.8
ARCOF
MOVL C00244 BC00244 V=166.7
SFTOF
MOVL C00245 BC00245 V=333.3
'------------------------
'W31.14
'------------------------
SFTON P0307
MOVL C00246 BC00246 V=333.3
MOVL C00247 BC00247 V=166.7 PL=0
ARCON
MOVL C00248 BC00248 V=10.8
ARCOF
MOVL C00249 BC00249 V=250.0
SFTOF
MOVL C00250 BC00250 V=500.0
MOVL C00251 BC00251 V=500.0
MOVJ C00252 BC00252 VJ=30.00
MOVJ C00253 BC00253 VJ=30.00
MOVJ C00254 BC00254 VJ=40.00
MOVJ C00255 BC00255 VJ=50.00
MOVJ C00256 BC00256 VJ=30.00
'------------------------
'W214A
'------------------------
SFTON P0351
MOVL C00257 BC00257 V=333.3
MOVL C00258 BC00258 V=500.0
MOVL C00259 BC00259 V=166.7 PL=0
MACRO1 MJ#(0) ARGF9
ARCON
MOVL C00260 BC00260 V=11.7
MOVL C00261 BC00261 V=11.3
ARCOF
SFTOF
MOVL C00262 BC00262 V=166.7
SFTOF
MOVJ C00263 BC00263 VJ=50.00
MOVJ C00264 BC00264 VJ=50.00
MOVJ C00265 BC00265 VJ=50.00
MOVJ C00266 BC00266 VJ=50.00
MOVJ C00267 BC00267 VJ=30.00
MOVJ C00268 BC00268 VJ=20.00
'------------------------
'W31.16
MACRO1 MJ#(0) ARGF10
'------------------------
SFTON P0308
MOVL C00269 BC00269 V=333.3
MOVL C00270 BC00270 V=133.3 PL=0
ARCON
MOVL C00271 BC00271 V=10.8
ARCOF
SFTOF
MOVL C00272 BC00272 V=250.0
SFTOF
'------------------------
'W31.18
'------------------------
SFTON P0309
MOVL C00273 BC00273 V=166.7
MOVL C00274 BC00274 V=166.7 PL=0
ARCON
MOVL C00275 BC00275 V=10.8
ARCOF
MOVL C00276 BC00276 V=166.7
SFTOF
'------------------------
'W31.19
'------------------------
SFTON P0310
MOVL C00277 BC00277 V=333.3
MOVL C00278 BC00278 V=166.7 PL=0
MACRO1 MJ#(0) ARGF10
ARCON
MOVL C00279 BC00279 V=10.8
ARCOF
MOVL C00280 BC00280 V=250.0
SFTOF
MOVL C00281 BC00281 V=250.0
MOVL C00282 BC00282 V=500.0
MOVL C00283 BC00283 V=666.7
MOVL C00284 BC00284 V=666.7
MOVJ C00285 BC00285 VJ=50.00
MOVJ C00286 BC00286 VJ=50.00
MOVJ C00287 BC00287 VJ=50.00
'------------------------
'W215A
'------------------------
SFTON P0359
MOVL C00288 BC00288 V=666.7
MOVL C00289 BC00289 V=166.7 PL=0
MACRO1 MJ#(0) ARGF9
ARCON
SFTOF
SFTON P0358
MOVL C00290 BC00290 V=11.7
ARCOF
MOVL C00291 BC00291 V=333.3
SFTOF
MOVJ C00292 BC00292 VJ=30.00
MOVJ C00293 BC00293 VJ=50.00
MOVJ C00294 BC00294 VJ=50.00
MOVJ C00295 BC00295 VJ=50.00
MOVJ C00296 BC00296 VJ=50.00
MOVJ C00297 BC00297 VJ=50.00
MOVJ C00298 BC00298 VJ=30.00
MOVJ C00299 BC00299 VJ=30.00
'------------------------
'W31.21
'------------------------
SFTON P0311
MOVL C00300 BC00300 V=666.7
MOVL C00301 BC00301 V=166.7 PL=0
MACRO1 MJ#(0) ARGF10
ARCON
MOVL C00302 BC00302 V=10.8
ARCOF
MOVL C00303 BC00303 V=250.0
SFTOF
'------------------------
'W31.22
'------------------------
SFTON P0312
MOVL C00304 BC00304 V=333.3
MOVL C00305 BC00305 V=166.7 PL=0
ARCON
MOVL C00306 BC00306 V=10.8
ARCOF
MOVL C00307 BC00307 V=250.0
SFTOF
'------------------------
'W31.24
'------------------------
SFTON P0313
MOVL C00308 BC00308 V=500.0
MOVL C00309 BC00309 V=166.7 PL=0
MACRO1 MJ#(0) ARGF10
ARCON
MOVL C00310 BC00310 V=10.8
ARCOF
SFTOF
MOVL C00311 BC00311 V=250.0
MOVL C00312 BC00312 V=333.3
MOVL C00313 BC00313 V=500.0
SFTOF
MOVJ C00314 BC00314 VJ=50.00
MOVJ C00315 BC00315 VJ=50.00
MOVJ C00316 BC00316 VJ=50.00
'::::::::::::::::::::::::
'::::::::::::::::::::::::
'::::::::::::::::::::::::
'::::::::::::::::::::::::
'::::::::::::::::::::::::
'::::::::::::::::::::::::
'::::::::::::::::::::::::
MOVJ C00317 BC00317 VJ=50.00
'------------------------
'W215A
'------------------------
MOVJ C00318 BC00318 VJ=80.00
MOVJ C00319 BC00319 VJ=80.00
COMM SFTON P0360
COMM MOVL C00320 BC00320 V=500.0
COMM MOVL C00321 BC00321 V=666.7
COMM MOVL C00322 BC00322 V=166.7 PL=0
COMM MACRO1 MJ#(0) ARGF9
COMM ARCON
COMM SFTOF
COMM SFTON P0361
COMM MOVL C00323 BC00323 V=11.7
COMM ARCOF
COMM MOVL C00324 BC00324 V=333.3
SFTOF
MOVJ C00325 BC00325 VJ=50.00
SFTON P0357
MOVL C00326 BC00326 V=666.7
MOVL C00327 BC00327 V=166.7 PL=0
MACRO1 MJ#(0) ARGF9
ARCON
SFTOF
SFTON P0356
MOVL C00328 BC00328 V=11.7
ARCOF
MOVL C00329 BC00329 V=333.3
MOVL C00330 BC00330 V=500.0
SFTOF
MOVJ C00331 BC00331 VJ=50.00
MOVJ C00332 BC00332 VJ=50.00
MOVJ C00333 BC00333 VJ=50.00
MOVJ C00334 BC00334 VJ=50.00
MOVJ C00335 BC00335 VJ=50.00
MOVJ C00336 BC00336 VJ=30.00
MOVL C00337 BC00337 V=666.7
'------------------------
'W31.29
'------------------------
SFTON P0316
MOVL C00338 BC00338 V=333.3
MOVL C00339 BC00339 V=333.3
MOVL C00340 BC00340 V=333.3
MOVL C00341 BC00341 V=66.7 PL=0
MACRO1 MJ#(0) ARGF10
ARCON
MOVL C00342 BC00342 V=10.8
ARCOF
MOVL C00343 BC00343 V=250.0
SFTOF
'------------------------
'W31.31
'------------------------
SFTON P0317
MOVL C00344 BC00344 V=666.7
MOVL C00345 BC00345 V=166.7 PL=0
ARCON
MOVL C00346 BC00346 V=10.8
ARCOF
SFTOF
MOVL C00347 BC00347 V=250.0
SFTOF
'------------------------
'W31.32
'------------------------
SFTON P0317
MOVL C00348 BC00348 V=333.3 PL=0
MOVL C00349 BC00349 V=166.7 PL=0
ARCON
MOVL C00350 BC00350 V=10.8
ARCOF
MOVL C00351 BC00351 V=250.0
SFTOF
MOVL C00352 BC00352 V=333.3
MOVL C00353 BC00353 V=333.3
MOVL C00354 BC00354 V=500.0
MOVL C00355 BC00355 V=500.0
MOVL C00356 BC00356 V=500.0
MOVJ C00357 BC00357 VJ=40.00
MOVJ C00358 BC00358 VJ=40.00
MOVJ C00359 BC00359 VJ=50.00
SFTON P0353
MOVL C00360 BC00360 V=500.0
MOVL C00361 BC00361 V=333.3
MOVL C00362 BC00362 V=166.7 PL=0
MACRO1 MJ#(0) ARGF9
ARCON
SFTOF
SFTON P0352
MOVL C00363 BC00363 V=11.7
ARCOF
MOVL C00364 BC00364 V=250.0
SFTOF
MOVJ C00365 BC00365 VJ=40.00
MOVJ C00366 BC00366 VJ=50.00
CALL JOB:FRONT_WELD_90ST-1_4040
CALL JOB:MOVE_OUT_OF_TUNNEL
END
